LIN {X 0,Y 202.903,Z 833.115,A -85,B 0,C 180,E1 -31559.988,E2 -31559.988} C_VEL
LIN {X 0,Y 208.884,Z 836.315,A -85,B 0,C 180,E1 -31563.074,E2 -31563.074} C_VEL
LIN {X 0,Y 216.378,Z 840.609,A -85,B 0,C 180,E1 -31567.061,E2 -31567.061} C_VEL
LIN {X 0,Y 220.572,Z 843.241,A -85,B 0,C 180,E1 -31569.483,E2 -31569.483} C_VEL
LIN {X 0,Y 224.304,Z 845.645,A -85,B 0,C 180,E1 -31571.741,E2 -31571.741} C_VEL
LIN {X 0,Y 227.405,Z 847.744,A -85,B 0,C 180,E1 -31573.851,E2 -31573.851} C_VEL
LIN {X 0,Y 230.992,Z 850.3,A -85,B 0,C 180,E1 -31576.804,E2 -31576.804} C_VEL
LIN {X 0,Y 235.032,Z 852.777,A -85,B 0,C 180,E1 -31580.667,E2 -31580.667} C_VEL
LIN {X 0,Y 237.24,Z 853.939,A -85,B 0,C 180,E1 -31583.195,E2 -31583.195} C_VEL
LIN {X 0,Y 238.369,Z 854.486,A -85,B 0,C 180,E1 -31584.926,E2 -31584.926} C_VEL
LIN {X 0,Y 239.315,Z 854.891,A -85,B 0,C 180,E1 -31586.829,E2 -31586.829} C_VEL
LIN {X 0,Y 239.828,Z 855.055,A -85,B 0,C 180,E1 -31588.321,E2 -31588.321} C_VEL
LIN {X 0,Y 240.028,Z 855.12,A -85,B 0,C 180,E1 -31590,E2 -31590} C_VEL
LIN {X 0,Y 239.805,Z 855.053,A -85,B 0,C 180,E1 -31591.679,E2 -31591.679} C_VEL
LIN {X 0,Y 239.195,Z 854.848,A -85,B 0,C 180,E1 -31593.369,E2 -31593.369} C_VEL
LIN {X 0,Y 238.362,Z 854.475,A -85,B 0,C 180,E1 -31595.075,E2 -31595.075} C_VEL
LIN {X 0,Y 237.219,Z 853.929,A -85,B 0,C 180,E1 -31596.806,E2 -31596.806} C_VEL
LIN {X 0,Y 235.033,Z 852.788,A -85,B 0,C 180,E1 -31599.335,E2 -31599.335} C_VEL
LIN {X 0,Y 230.986,Z 850.298,A -85,B 0,C 180,E1 -31603.19,E2 -31603.19} C_VEL
LIN {X 0,Y 227.067,Z 847.531,A -85,B 0,C 180,E1 -31606.368,E2 -31606.368} C_VEL
LIN {X 0,Y 223.04,Z 844.829,A -85,B 0,C 180,E1 -31609.041,E2 -31609.041} C_VEL
LIN {X 0,Y 220.517,Z 843.221,A -85,B 0,C 180,E1 -31610.538,E2 -31610.538} C_VEL
LIN {X 0,Y 217.608,Z 841.994,A -85,B 0,C 180,E1 -31611.838,E2 -31611.838} C_VEL
LIN {X 0,Y 213.839,Z 841.077,A -85,B 0,C 180,E1 -31613.032,E2 -31613.032} C_VEL
LIN {X 0,Y 203.07,Z 838.775,A -85,B 0,C 180,E1 -31616.24,E2 -31616.24} C_VEL
LIN {X 0,Y 200.951,Z 837.913,A -85,B 0,C 180,E1 -31617.173,E2 -31617.173} C_VEL
LIN {X 0,Y 194.952,Z 834.972,A -85,B 0,C 180,E1 -31620.31,E2 -31620.31} C_VEL
LIN {X 0,Y 187.377,Z 831.364,A -85,B 0,C 180,E1 -31624.397,E2 -31624.397} C_VEL
LIN {X 0,Y 176.623,Z 826.157,A -85,B 0,C 180,E1 -31630.886,E2 -31630.886} C_VEL
LIN {X 0,Y 162.798,Z 817.399,A -85,B 0,C 180,E1 -31642.817,E2 -31642.817} C_VEL
LIN {X 0,Y 160.588,Z 818.703,A -85,B 0,C 180,E1 -31642.859,E2 -31642.859} C_VEL
LIN {X 0,Y 146.717,Z 829.238,A -85,B 0,C 180,E1 -31640.033,E2 -31640.033} C_VEL
LIN {X 0,Y 134.403,Z 837.203,A -85,B 0,C 180,E1 -31637.058,E2 -31637.058} C_VEL
LIN {X 0,Y 122.45,Z 843.857,A -85,B 0,C 180,E1 -31633.529,E2 -31633.529} C_VEL
LIN {X 0,Y 111.056,Z 849.379,A -85,B 0,C 180,E1 -31629.258,E2 -31629.258} C_VEL
LIN {X 0,Y 100.44,Z 853.782,A -85,B 0,C 180,E1 -31624.039,E2 -31624.039} C_VEL
LIN {X 0,Y 90.867,Z 857.174,A -85,B 0,C 180,E1 -31617.649,E2 -31617.649} C_VEL
LIN {X 0,Y 81.549,Z 859.864,A -85,B 0,C 180,E1 -31608.564,E2 -31608.564} C_VEL
LIN {X 0,Y 76.46,Z 861.04,A -85,B 0,C 180,E1 -31600.593,E2 -31600.593} C_VEL
LIN {X 0,Y 72.976,Z 861.583,A -85,B 0,C 180,E1 -31590,E2 -31590} C_VEL
LIN {X 0,Y 76.461,Z 861.04,A -85,B 0,C 180,E1 -31579.407,E2 -31579.407} C_VEL
LIN {X 0,Y 82.645,Z 859.587,A -85,B 0,C 180,E1 -31570.114,E2 -31570.114} C_VEL
LIN {X 0,Y 90.866,Z 857.173,A -85,B 0,C 180,E1 -31562.351,E2 -31562.351} C_VEL
LIN {X 0,Y 100.444,Z 853.782,A -85,B 0,C 180,E1 -31555.962,E2 -31555.962} C_VEL
LIN {X 0,Y 111.054,Z 849.379,A -85,B 0,C 180,E1 -31550.741,E2 -31550.741} C_VEL
LIN {X 0,Y 122.424,Z 843.858,A -85,B 0,C 180,E1 -31546.459,E2 -31546.459} C_VEL
LIN {X 0,Y 134.403,Z 837.203,A -85,B 0,C 180,E1 -31542.941,E2 -31542.941} C_VEL
LIN {X 0,Y 146.733,Z 829.238,A -85,B 0,C 180,E1 -31539.975,E2 -31539.975} C_VEL
LIN {X 0,Y 160.605,Z 818.703,A -85,B 0,C 180,E1 -31537.149,E2 -31537.149} C_VEL
LIN {X 0,Y 162.798,Z 817.399,A -85,B 0,C 180,E1 -31537.183,E2 -31537.183} C_VEL
LIN {X 0,Y 176.609,Z 826.17,A -85,B 0,C 180,E1 -31549.119,E2 -31549.119} C_VEL
LIN {X 0,Y 187.851,Z 831.576,A -85,B 0,C 180,E1 -31555.863,E2 -31555.863} C_VEL
LIN {X 0,Y 195.144,Z 835.087,A -85,B 0,C 180,E1 -31559.806,E2 -31559.806} C_VEL
LIN {X 0,Y 201.261,Z 838.095,A -85,B 0,C 180,E1 -31563.003,E2 -31563.003} C_VEL
LIN {X 0,Y 209.419,Z 842.368,A -85,B 0,C 180,E1 -31567.349,E2 -31567.349} C_VEL
LIN {X 0,Y 215.586,Z 845.919,A -85,B 0,C 180,E1 -31570.975,E2 -31570.975} C_VEL
LIN {X 0,Y 219.709,Z 848.454,A -85,B 0,C 180,E1 -31573.662,E2 -31573.662} C_VEL
LIN {X 0,Y 224.303,Z 851.529,A -85,B 0,C 180,E1 -31577.331,E2 -31577.331} C_VEL
LIN {X 0,Y 227.865,Z 853.75,A -85,B 0,C 180,E1 -31580.736,E2 -31580.736} C_VEL
LIN {X 0,Y 229.868,Z 854.802,A -85,B 0,C 180,E1 -31582.976,E2 -31582.976} C_VEL
LIN {X 0,Y 231.161,Z 855.444,A -85,B 0,C 180,E1 -31584.767,E2 -31584.767} C_VEL
LIN {X 0,Y 232.263,Z 855.927,A -85,B 0,C 180,E1 -31586.891,E2 -31586.891} C_VEL
LIN {X 0,Y 232.778,Z 856.084,A -85,B 0,C 180,E1 -31588.27,E2 -31588.27} C_VEL
LIN {X 0,Y 233.006,Z 856.158,A -85,B 0,C 180,E1 -31590,E2 -31590} C_VEL
LIN {X 0,Y 232.759,Z 856.085,A -85,B 0,C 180,E1 -31591.73,E2 -31591.73} C_VEL
LIN {X 0,Y 232.081,Z 855.86,A -85,B 0,C 180,E1 -31593.472,E2 -31593.472} C_VEL
LIN {X 0,Y 231.152,Z 855.444,A -85,B 0,C 180,E1 -31595.233,E2 -31595.233} C_VEL
LIN {X 0,Y 229.854,Z 854.809,A -85,B 0,C 180,E1 -31597.025,E2 -31597.025} C_VEL
LIN {X 0,Y 227.867,Z 853.762,A -85,B 0,C 180,E1 -31599.267,E2 -31599.267} C_VEL
LIN {X 0,Y 224.289,Z 851.528,A -85,B 0,C 180,E1 -31602.67,E2 -31602.67} C_VEL
LIN {X 0,Y 219.695,Z 848.469,A -85,B 0,C 180,E1 -31606.326,E2 -31606.326} C_VEL
LIN {X 0,Y 215.549,Z 845.92,A -85,B 0,C 180,E1 -31609.029,E2 -31609.029} C_VEL
LIN {X 0,Y 209.405,Z 842.382,A -85,B 0,C 180,E1 -31612.641,E2 -31612.641} C_VEL
LIN {X 0,Y 200.951,Z 837.913,A -85,B 0,C 180,E1 -31617.173,E2 -31617.173} C_VEL
LIN {X 0,Y 197.626,Z 836.788,A -85,B 0,C 180,E1 -31618.533,E2 -31618.533} C_VEL
LIN {X 0,Y 190.664,Z 835.781,A -85,B 0,C 180,E1 -31620.593,E2 -31620.593} C_VEL
LIN {X 0,Y 184.942,Z 835.104,A -85,B 0,C 180,E1 -31622.296,E2 -31622.296} C_VEL
LIN {X 0,Y 181.269,Z 834.289,A -85,B 0,C 180,E1 -31623.747,E2 -31623.747} C_VEL
LIN {X 0,Y 180.266,Z 833.88,A -85,B 0,C 180,E1 -31624.278,E2 -31624.278} C_VEL
LIN {X 0,Y 172.251,Z 830.257,A -85,B 0,C 180,E1 -31629.177,E2 -31629.177} C_VEL
LIN {X 0,Y 159.808,Z 823.458,A -85,B 0,C 180,E1 -31639.177,E2 -31639.177} C_VEL
LIN {X 0,Y 157.5,Z 824.5,A -85,B 0,C 180,E1 -31639.338,E2 -31639.338} C_VEL
LIN {X 0,Y 145.363,Z 833.226,A -85,B 0,C 180,E1 -31636.486,E2 -31636.486} C_VEL
LIN {X 0,Y 133.54,Z 840.53,A -85,B 0,C 180,E1 -31633.169,E2 -31633.169} C_VEL
LIN {X 0,Y 122.185,Z 846.563,A -85,B 0,C 180,E1 -31629.249,E2 -31629.249} C_VEL
LIN {X 0,Y 109.682,Z 852.261,A -85,B 0,C 180,E1 -31623.595,E2 -31623.595} C_VEL
LIN {X 0,Y 97.33,Z 856.961,A -85,B 0,C 180,E1 -31615.673,E2 -31615.673} C_VEL
LIN {X 0,Y 87.937,Z 859.783,A -85,B 0,C 180,E1 -31606.458,E2 -31606.458} C_VEL
LIN {X 0,Y 83.554,Z 860.825,A -85,B 0,C 180,E1 -31599.684,E2 -31599.684} C_VEL
LIN {X 0,Y 80.137,Z 861.372,A -85,B 0,C 180,E1 -31590,E2 -31590} C_VEL
LIN {X 0,Y 83.555,Z 860.825,A -85,B 0,C 180,E1 -31580.316,E2 -31580.316} C_VEL
LIN {X 0,Y 89.45,Z 859.373,A -85,B 0,C 180,E1 -31571.683,E2 -31571.683} C_VEL
LIN {X 0,Y 97.33,Z 856.961,A -85,B 0,C 180,E1 -31564.327,E2 -31564.327} C_VEL
LIN {X 0,Y 109.68,Z 852.262,A -85,B 0,C 180,E1 -31556.406,E2 -31556.406} C_VEL
LIN {X 0,Y 122.173,Z 846.563,A -85,B 0,C 180,E1 -31550.746,E2 -31550.746} C_VEL
LIN {X 0,Y 136.64,Z 838.692,A -85,B 0,C 180,E1 -31545.901,E2 -31545.901} C_VEL
LIN {X 0,Y 148.422,Z 831.14,A -85,B 0,C 180,E1 -31542.783,E2 -31542.783} C_VEL
LIN {X 0,Y 157.533,Z 824.499,A -85,B 0,C 180,E1 -31540.677,E2 -31540.677} C_VEL
LIN {X 0,Y 159.823,Z 823.457,A -85,B 0,C 180,E1 -31540.829,E2 -31540.829} C_VEL
LIN {X 0,Y 172.239,Z 830.268,A -85,B 0,C 180,E1 -31550.828,E2 -31550.828} C_VEL
LIN {X 0,Y 183.391,Z 835.249,A -85,B 0,C 180,E1 -31557.467,E2 -31557.467} C_VEL
LIN {X 0,Y 191.402,Z 838.842,A -85,B 0,C 180,E1 -31561.791,E2 -31561.791} C_VEL
LIN {X 0,Y 196.719,Z 841.243,A -85,B 0,C 180,E1 -31564.615,E2 -31564.615} C_VEL
LIN {X 0,Y 203.902,Z 844.75,A -85,B 0,C 180,E1 -31568.53,E2 -31568.53} C_VEL
LIN {X 0,Y 208.106,Z 846.961,A -85,B 0,C 180,E1 -31571.011,E2 -31571.011} C_VEL
LIN {X 0,Y 212.316,Z 849.306,A -85,B 0,C 180,E1 -31573.726,E2 -31573.726} C_VEL
LIN {X 0,Y 216.441,Z 851.835,A -85,B 0,C 180,E1 -31576.934,E2 -31576.934} C_VEL
LIN {X 0,Y 218.611,Z 853.231,A -85,B 0,C 180,E1 -31578.879,E2 -31578.879} C_VEL
LIN {X 0,Y 220.68,Z 854.365,A -85,B 0,C 180,E1 -31580.838,E2 -31580.838} C_VEL
LIN {X 0,Y 222.416,Z 855.312,A -85,B 0,C 180,E1 -31582.739,E2 -31582.739} C_VEL
LIN {X 0,Y 223.851,Z 856.031,A -85,B 0,C 180,E1 -31584.596,E2 -31584.596} C_VEL
LIN {X 0,Y 225.207,Z 856.635,A -85,B 0,C 180,E1 -31586.975,E2 -31586.975} C_VEL
LIN {X 0,Y 225.66,Z 856.792,A -85,B 0,C 180,E1 -31588.215,E2 -31588.215} C_VEL
LIN {X 0,Y 225.935,Z 856.875,A -85,B 0,C 180,E1 -31590,E2 -31590} C_VEL
LIN {X 0,Y 225.644,Z 856.796,A -85,B 0,C 180,E1 -31591.785,E2 -31591.785} C_VEL
LIN {X 0,Y 224.902,Z 856.532,A -85,B 0,C 180,E1 -31593.583,E2 -31593.583} C_VEL
LIN {X 0,Y 223.842,Z 856.039,A -85,B 0,C 180,E1 -31595.405,E2 -31595.405} C_VEL
LIN {X 0,Y 222.405,Z 855.308,A -85,B 0,C 180,E1 -31597.261,E2 -31597.261} C_VEL
LIN {X 0,Y 220.68,Z 854.366,A -85,B 0,C 180,E1 -31599.162,E2 -31599.162} C_VEL
LIN {X 0,Y 218.613,Z 853.231,A -85,B 0,C 180,E1 -31601.121,E2 -31601.121} C_VEL
LIN {X 0,Y 216.341,Z 851.781,A -85,B 0,C 180,E1 -31603.144,E2 -31603.144} C_VEL
LIN {X 0,Y 212.307,Z 849.314,A -85,B 0,C 180,E1 -31606.266,E2 -31606.266} C_VEL
LIN {X 0,Y 208.098,Z 846.969,A -85,B 0,C 180,E1 -31608.983,E2 -31608.983} C_VEL
LIN {X 0,Y 202.014,Z 843.832,A -85,B 0,C 180,E1 -31612.5,E2 -31612.5} C_VEL
LIN {X 0,Y 194.896,Z 840.388,A -85,B 0,C 180,E1 -31616.354,E2 -31616.354} C_VEL
LIN {X 0,Y 187.335,Z 836.998,A -85,B 0,C 180,E1 -31620.362,E2 -31620.362} C_VEL
LIN {X 0,Y 180.266,Z 833.88,A -85,B 0,C 180,E1 -31624.278,E2 -31624.278} C_VEL
LIN {X 0,Y 176.99,Z 832.953,A -85,B 0,C 180,E1 -31625.821,E2 -31625.821} C_VEL
LIN {X 0,Y 170.275,Z 832.301,A -85,B 0,C 180,E1 -31628.215,E2 -31628.215} C_VEL
LIN {X 0,Y 164.882,Z 831.868,A -85,B 0,C 180,E1 -31630.224,E2 -31630.224} C_VEL
LIN {X 0,Y 161.52,Z 831.172,A -85,B 0,C 180,E1 -31631.928,E2 -31631.928} C_VEL
LIN {X 0,Y 160.634,Z 830.815,A -85,B 0,C 180,E1 -31632.546,E2 -31632.546} C_VEL
LIN {X 0,Y 156.751,Z 828.796,A -85,B 0,C 180,E1 -31635.836,E2 -31635.836} C_VEL
LIN {X 0,Y 156.312,Z 828.815,A -85,B 0,C 180,E1 -31636.002,E2 -31636.002} C_VEL
LIN {X 0,Y 144.598,Z 836.785,A -85,B 0,C 180,E1 -31632.878,E2 -31632.878} C_VEL
LIN {X 0,Y 133.295,Z 843.432,A -85,B 0,C 180,E1 -31629.249,E2 -31629.249} C_VEL
LIN {X 0,Y 122.573,Z 848.958,A -85,B 0,C 180,E1 -31624.985,E2 -31624.985} C_VEL
LIN {X 0,Y 112.704,Z 853.353,A -85,B 0,C 180,E1 -31619.924,E2 -31619.924} C_VEL
LIN {X 0,Y 103.892,Z 856.748,A -85,B 0,C 180,E1 -31613.946,E2 -31613.946} C_VEL
LIN {X 0,Y 94.435,Z 859.688,A -85,B 0,C 180,E1 -31604.657,E2 -31604.657} C_VEL
LIN {X 0,Y 88.689,Z 860.946,A -85,B 0,C 180,E1 -31594.545,E2 -31594.545} C_VEL
LIN {X 0,Y 87.31,Z 861.16,A -85,B 0,C 180,E1 -31590,E2 -31590} C_VEL
LIN {X 0,Y 90.667,Z 860.611,A -85,B 0,C 180,E1 -31581.082,E2 -31581.082} C_VEL
LIN {X 0,Y 96.321,Z 859.158,A -85,B 0,C 180,E1 -31573.031,E2 -31573.031} C_VEL
LIN {X 0,Y 103.893,Z 856.748,A -85,B 0,C 180,E1 -31566.054,E2 -31566.054} C_VEL
LIN {X 0,Y 115.065,Z 852.356,A -85,B 0,C 180,E1 -31558.768,E2 -31558.768} C_VEL
LIN {X 0,Y 125.186,Z 847.669,A -85,B 0,C 180,E1 -31553.881,E2 -31553.881} C_VEL
LIN {X 0,Y 136.047,Z 841.889,A -85,B 0,C 180,E1 -31549.781,E2 -31549.781} C_VEL
LIN {X 0,Y 147.492,Z 834.947,A -85,B 0,C 180,E1 -31546.298,E2 -31546.298} C_VEL
LIN {X 0,Y 156.329,Z 828.814,A -85,B 0,C 180,E1 -31544.004,E2 -31544.004} C_VEL
LIN {X 0,Y 156.733,Z 828.797,A -85,B 0,C 180,E1 -31544.157,E2 -31544.157} C_VEL
LIN {X 0,Y 167.935,Z 834.178,A -85,B 0,C 180,E1 -31552.667,E2 -31552.667} C_VEL
LIN {X 0,Y 175.515,Z 837.267,A -85,B 0,C 180,E1 -31557.232,E2 -31557.232} C_VEL
LIN {X 0,Y 183.577,Z 840.555,A -85,B 0,C 180,E1 -31561.704,E2 -31561.704} C_VEL
LIN {X 0,Y 187.76,Z 842.305,A -85,B 0,C 180,E1 -31563.938,E2 -31563.938} C_VEL
LIN {X 0,Y 192.07,Z 844.153,A -85,B 0,C 180,E1 -31566.266,E2 -31566.266} C_VEL
LIN {X 0,Y 197.335,Z 846.497,A -85,B 0,C 180,E1 -31569.137,E2 -31569.137} C_VEL
LIN {X 0,Y 201.689,Z 848.569,A -85,B 0,C 180,E1 -31571.723,E2 -31571.723} C_VEL
LIN {X 0,Y 205.35,Z 850.388,A -85,B 0,C 180,E1 -31574.11,E2 -31574.11} C_VEL
LIN {X 0,Y 209.141,Z 852.488,A -85,B 0,C 180,E1 -31577.034,E2 -31577.034} C_VEL
LIN {X 0,Y 210.783,Z 853.466,A -85,B 0,C 180,E1 -31578.46,E2 -31578.46} C_VEL
LIN {X 0,Y 213.479,Z 854.859,A -85,B 0,C 180,E1 -31580.976,E2 -31580.976} C_VEL
LIN {X 0,Y 214.893,Z 855.555,A -85,B 0,C 180,E1 -31582.483,E2 -31582.483} C_VEL
LIN {X 0,Y 216.462,Z 856.339,A -85,B 0,C 180,E1 -31584.411,E2 -31584.411} C_VEL
LIN {X 0,Y 218.14,Z 857.02,A -85,B 0,C 180,E1 -31587.121,E2 -31587.121} C_VEL
LIN {X 0,Y 218.854,Z 857.272,A -85,B 0,C 180,E1 -31590,E2 -31590} C_VEL
LIN {X 0,Y 218.136,Z 857.025,A -85,B 0,C 180,E1 -31592.858,E2 -31592.858} C_VEL
LIN {X 0,Y 216.453,Z 856.339,A -85,B 0,C 180,E1 -31595.59,E2 -31595.59} C_VEL
LIN {X 0,Y 214.887,Z 855.556,A -85,B 0,C 180,E1 -31597.517,E2 -31597.517} C_VEL
LIN {X 0,Y 212.969,Z 854.598,A -85,B 0,C 180,E1 -31599.497,E2 -31599.497} C_VEL
LIN {X 0,Y 210.783,Z 853.466,A -85,B 0,C 180,E1 -31601.54,E2 -31601.54} C_VEL
LIN {X 0,Y 208.237,Z 852.026,A -85,B 0,C 180,E1 -31603.665,E2 -31603.665} C_VEL
LIN {X 0,Y 204.905,Z 850.162,A -85,B 0,C 180,E1 -31606.188,E2 -31606.188} C_VEL
LIN {X 0,Y 200.599,Z 848.03,A -85,B 0,C 180,E1 -31608.927,E2 -31608.927} C_VEL
LIN {X 0,Y 196.286,Z 846.05,A -85,B 0,C 180,E1 -31611.422,E2 -31611.422} C_VEL
LIN {X 0,Y 191.988,Z 844.124,A -85,B 0,C 180,E1 -31613.774,E2 -31613.774} C_VEL
LIN {X 0,Y 186.112,Z 841.59,A -85,B 0,C 180,E1 -31616.945,E2 -31616.945} C_VEL
LIN {X 0,Y 179.298,Z 838.839,A -85,B 0,C 180,E1 -31620.634,E2 -31620.634} C_VEL
LIN {X 0,Y 171.662,Z 835.698,A -85,B 0,C 180,E1 -31625.035,E2 -31625.035} C_VEL
LIN {X 0,Y 160.634,Z 830.815,A -85,B 0,C 180,E1 -31632.546,E2 -31632.546} C_VEL
LIN {X 0,Y 159.568,Z 830.875,A -85,B 0,C 180,E1 -31632.887,E2 -31632.887} C_VEL
LIN {X 0,Y 157.126,Z 831.782,A -85,B 0,C 180,E1 -31632.998,E2 -31632.998} C_VEL
LIN {X 0,Y 153.935,Z 833.506,A -85,B 0,C 180,E1 -31632.595,E2 -31632.595} C_VEL
LIN {X 0,Y 148.459,Z 837.36,A -85,B 0,C 180,E1 -31630.799,E2 -31630.799} C_VEL
LIN {X 0,Y 143.925,Z 840.362,A -85,B 0,C 180,E1 -31629.105,E2 -31629.105} C_VEL
LIN {X 0,Y 133.687,Z 846.134,A -85,B 0,C 180,E1 -31625.328,E2 -31625.328} C_VEL
LIN {X 0,Y 123.661,Z 851.081,A -85,B 0,C 180,E1 -31620.763,E2 -31620.763} C_VEL
LIN {X 0,Y 114.61,Z 854.929,A -85,B 0,C 180,E1 -31615.419,E2 -31615.419} C_VEL
LIN {X 0,Y 106.713,Z 857.827,A -85,B 0,C 180,E1 -31609.225,E2 -31609.225} C_VEL
LIN {X 0,Y 100.286,Z 859.76,A -85,B 0,C 180,E1 -31602.136,E2 -31602.136} C_VEL
LIN {X 0,Y 95.842,Z 860.737,A -85,B 0,C 180,E1 -31594.205,E2 -31594.205} C_VEL
LIN {X 0,Y 94.494,Z 860.947,A -85,B 0,C 180,E1 -31590,E2 -31590} C_VEL
LIN {X 0,Y 97.796,Z 860.396,A -85,B 0,C 180,E1 -31581.737,E2 -31581.737} C_VEL
LIN {X 0,Y 103.268,Z 858.942,A -85,B 0,C 180,E1 -31574.204,E2 -31574.204} C_VEL
LIN {X 0,Y 110.534,Z 856.536,A -85,B 0,C 180,E1 -31567.574,E2 -31567.574} C_VEL
LIN {X 0,Y 120.694,Z 852.41,A -85,B 0,C 180,E1 -31560.86,E2 -31560.86} C_VEL
LIN {X 0,Y 131.092,Z 847.459,A -85,B 0,C 180,E1 -31555.743,E2 -31555.743} C_VEL
LIN {X 0,Y 141.642,Z 841.678,A -85,B 0,C 180,E1 -31551.669,E2 -31551.669} C_VEL
LIN {X 0,Y 152.464,Z 834.953,A -85,B 0,C 180,E1 -31548.26,E2 -31548.26} C_VEL
LIN {X 0,Y 154.544,Z 833.994,A -85,B 0,C 180,E1 -31548.109,E2 -31548.109} C_VEL
LIN {X 0,Y 167.591,Z 839.291,A -85,B 0,C 180,E1 -31557.002,E2 -31557.002} C_VEL
LIN {X 0,Y 175.719,Z 842.283,A -85,B 0,C 180,E1 -31561.629,E2 -31561.629} C_VEL
LIN {X 0,Y 181.627,Z 844.494,A -85,B 0,C 180,E1 -31564.809,E2 -31564.809} C_VEL
LIN {X 0,Y 188.623,Z 847.294,A -85,B 0,C 180,E1 -31568.665,E2 -31568.665} C_VEL
LIN {X 0,Y 193.066,Z 849.118,A -85,B 0,C 180,E1 -31571.162,E2 -31571.162} C_VEL
LIN {X 0,Y 197.474,Z 851.04,A -85,B 0,C 180,E1 -31573.925,E2 -31573.925} C_VEL
LIN {X 0,Y 201.831,Z 853.152,A -85,B 0,C 180,E1 -31577.156,E2 -31577.156} C_VEL
LIN {X 0,Y 206.282,Z 855.342,A -85,B 0,C 180,E1 -31581.119,E2 -31581.119} C_VEL
LIN {X 0,Y 209.018,Z 856.557,A -85,B 0,C 180,E1 -31584.211,E2 -31584.211} C_VEL
LIN {X 0,Y 211.075,Z 857.269,A -85,B 0,C 180,E1 -31587.276,E2 -31587.276} C_VEL
LIN {X 0,Y 211.75,Z 857.482,A -85,B 0,C 180,E1 -31590,E2 -31590} C_VEL
LIN {X 0,Y 211.072,Z 857.271,A -85,B 0,C 180,E1 -31592.706,E2 -31592.706} C_VEL
LIN {X 0,Y 209.011,Z 856.557,A -85,B 0,C 180,E1 -31595.789,E2 -31595.789} C_VEL
LIN {X 0,Y 206.282,Z 855.343,A -85,B 0,C 180,E1 -31598.881,E2 -31598.881} C_VEL
LIN {X 0,Y 201.828,Z 853.156,A -85,B 0,C 180,E1 -31602.84,E2 -31602.84} C_VEL
LIN {X 0,Y 197.467,Z 851.047,A -85,B 0,C 180,E1 -31606.068,E2 -31606.068} C_VEL
LIN {X 0,Y 192.398,Z 848.861,A -85,B 0,C 180,E1 -31609.193,E2 -31609.193} C_VEL
LIN {X 0,Y 187.349,Z 846.817,A -85,B 0,C 180,E1 -31612.032,E2 -31612.032} C_VEL
LIN {X 0,Y 179.979,Z 843.878,A -85,B 0,C 180,E1 -31616.089,E2 -31616.089} C_VEL
LIN {X 0,Y 171.585,Z 840.751,A -85,B 0,C 180,E1 -31620.669,E2 -31620.669} C_VEL
LIN {X 0,Y 163.737,Z 837.799,A -85,B 0,C 180,E1 -31625.362,E2 -31625.362} C_VEL
LIN {X 0,Y 154.544,Z 833.987,A -85,B 0,C 180,E1 -31631.897,E2 -31631.897} C_VEL
LIN {X 0,Y 152.464,Z 834.942,A -85,B 0,C 180,E1 -31631.75,E2 -31631.75} C_VEL
LIN {X 0,Y 143.925,Z 840.362,A -85,B 0,C 180,E1 -31629.105,E2 -31629.105} C_VEL
LIN {X 0,Y 140.3,Z 842.755,A -85,B 0,C 180,E1 -31627.479,E2 -31627.479} C_VEL
LIN {X 0,Y 132.687,Z 849.09,A -85,B 0,C 180,E1 -31621.236,E2 -31621.236} C_VEL
LIN {X 0,Y 129.812,Z 850.892,A -85,B 0,C 180,E1 -31619.127,E2 -31619.127} C_VEL
LIN {X 0,Y 128.668,Z 851.442,A -85,B 0,C 180,E1 -31618.463,E2 -31618.463} C_VEL
LIN {X 0,Y 117.24,Z 856.323,A -85,B 0,C 180,E1 -31611.08,E2 -31611.08} C_VEL
LIN {X 0,Y 110.272,Z 858.726,A -85,B 0,C 180,E1 -31604.769,E2 -31604.769} C_VEL
LIN {X 0,Y 104.932,Z 860.182,A -85,B 0,C 180,E1 -31597.698,E2 -31597.698} C_VEL
LIN {X 0,Y 101.676,Z 860.735,A -85,B 0,C 180,E1 -31590,E2 -31590} C_VEL
LIN {X 0,Y 104.932,Z 860.182,A -85,B 0,C 180,E1 -31582.302,E2 -31582.302} C_VEL
LIN {X 0,Y 110.223,Z 858.727,A -85,B 0,C 180,E1 -31575.224,E2 -31575.224} C_VEL
LIN {X 0,Y 117.242,Z 856.323,A -85,B 0,C 180,E1 -31568.921,E2 -31568.921} C_VEL
LIN {X 0,Y 126.463,Z 852.464,A -85,B 0,C 180,E1 -31562.768,E2 -31562.768} C_VEL
LIN {X 0,Y 137.111,Z 847.249,A -85,B 0,C 180,E1 -31557.439,E2 -31557.439} C_VEL
LIN {X 0,Y 147.367,Z 841.466,A -85,B 0,C 180,E1 -31553.408,E2 -31553.408} C_VEL
LIN {X 0,Y 151.841,Z 838.728,A -85,B 0,C 180,E1 -31551.89,E2 -31551.89} C_VEL
LIN {X 0,Y 155.78,Z 839.883,A -85,B 0,C 180,E1 -31554.297,E2 -31554.297} C_VEL
LIN {X 0,Y 163.634,Z 842.573,A -85,B 0,C 180,E1 -31559.202,E2 -31559.202} C_VEL
LIN {X 0,Y 172.116,Z 845.419,A -85,B 0,C 180,E1 -31563.937,E2 -31563.937} C_VEL
LIN {X 0,Y 177.015,Z 847.147,A -85,B 0,C 180,E1 -31566.608,E2 -31566.608} C_VEL
LIN {X 0,Y 182.696,Z 849.168,A -85,B 0,C 180,E1 -31569.745,E2 -31569.745} C_VEL
LIN {X 0,Y 187.573,Z 850.939,A -85,B 0,C 180,E1 -31572.558,E2 -31572.558} C_VEL
LIN {X 0,Y 191.545,Z 852.533,A -85,B 0,C 180,E1 -31575.118,E2 -31575.118} C_VEL
LIN {X 0,Y 194.781,Z 853.947,A -85,B 0,C 180,E1 -31577.497,E2 -31577.497} C_VEL
LIN {X 0,Y 199.077,Z 855.79,A -85,B 0,C 180,E1 -31581.29,E2 -31581.29} C_VEL
LIN {X 0,Y 201.541,Z 856.776,A -85,B 0,C 180,E1 -31583.995,E2 -31583.995} C_VEL
LIN {X 0,Y 204.005,Z 857.506,A -85,B 0,C 180,E1 -31587.489,E2 -31587.489} C_VEL
LIN {X 0,Y 204.644,Z 857.692,A -85,B 0,C 180,E1 -31590,E2 -31590} C_VEL
LIN {X 0,Y 204.002,Z 857.507,A -85,B 0,C 180,E1 -31592.494,E2 -31592.494} C_VEL
LIN {X 0,Y 201.536,Z 856.776,A -85,B 0,C 180,E1 -31596.005,E2 -31596.005} C_VEL
LIN {X 0,Y 199.077,Z 855.79,A -85,B 0,C 180,E1 -31598.71,E2 -31598.71} C_VEL
LIN {X 0,Y 194.507,Z 853.832,A -85,B 0,C 180,E1 -31602.693,E2 -31602.693} C_VEL
LIN {X 0,Y 190.02,Z 851.935,A -85,B 0,C 180,E1 -31605.927,E2 -31605.927} C_VEL
LIN {X 0,Y 185.459,Z 850.174,A -85,B 0,C 180,E1 -31608.672,E2 -31608.672} C_VEL
LIN {X 0,Y 180.937,Z 848.522,A -85,B 0,C 180,E1 -31611.22,E2 -31611.22} C_VEL
LIN {X 0,Y 176.511,Z 846.946,A -85,B 0,C 180,E1 -31613.686,E2 -31613.686} C_VEL
LIN {X 0,Y 167.825,Z 844.012,A -85,B 0,C 180,E1 -31618.43,E2 -31618.43} C_VEL
LIN {X 0,Y 159.624,Z 841.188,A -85,B 0,C 180,E1 -31623.225,E2 -31623.225} C_VEL
LIN {X 0,Y 155.311,Z 839.692,A -85,B 0,C 180,E1 -31626.033,E2 -31626.033} C_VEL
LIN {X 0,Y 151.845,Z 838.726,A -85,B 0,C 180,E1 -31628.111,E2 -31628.111} C_VEL
LIN {X 0,Y 139.643,Z 845.92,A -85,B 0,C 180,E1 -31623.614,E2 -31623.614} C_VEL
LIN {X 0,Y 128.668,Z 851.442,A -85,B 0,C 180,E1 -31618.463,E2 -31618.463} C_VEL
LIN {X 0,Y 125.679,Z 853.079,A -85,B 0,C 180,E1 -31616.28,E2 -31616.28} C_VEL
LIN {X 0,Y 122.718,Z 855.332,A -85,B 0,C 180,E1 -31612.04,E2 -31612.04} C_VEL
LIN {X 0,Y 120.934,Z 856.879,A -85,B 0,C 180,E1 -31608.47,E2 -31608.47} C_VEL
LIN {X 0,Y 119.134,Z 857.844,A -85,B 0,C 180,E1 -31605.825,E2 -31605.825} C_VEL
LIN {X 0,Y 118.339,Z 858.125,A -85,B 0,C 180,E1 -31604.968,E2 -31604.968} C_VEL
LIN {X 0,Y 112.067,Z 859.968,A -85,B 0,C 180,E1 -31597.205,E2 -31597.205} C_VEL
LIN {X 0,Y 108.856,Z 860.523,A -85,B 0,C 180,E1 -31590,E2 -31590} C_VEL
LIN {X 0,Y 112.068,Z 859.968,A -85,B 0,C 180,E1 -31582.795,E2 -31582.795} C_VEL
LIN {X 0,Y 117.226,Z 858.512,A -85,B 0,C 180,E1 -31576.125,E2 -31576.125} C_VEL
LIN {X 0,Y 124,Z 856.111,A -85,B 0,C 180,E1 -31570.12,E2 -31570.12} C_VEL
LIN {X 0,Y 132.346,Z 852.511,A -85,B 0,C 180,E1 -31564.521,E2 -31564.521} C_VEL
LIN {X 0,Y 143.255,Z 847.038,A -85,B 0,C 180,E1 -31558.995,E2 -31558.995} C_VEL
LIN {X 0,Y 150.76,Z 842.793,A -85,B 0,C 180,E1 -31555.986,E2 -31555.986} C_VEL
LIN {X 0,Y 159.858,Z 845.637,A -85,B 0,C 180,E1 -31561.553,E2 -31561.553} C_VEL
LIN {X 0,Y 166.026,Z 847.501,A -85,B 0,C 180,E1 -31564.957,E2 -31564.957} C_VEL
LIN {X 0,Y 173.229,Z 849.746,A -85,B 0,C 180,E1 -31568.924,E2 -31568.924} C_VEL
LIN {X 0,Y 177.995,Z 851.238,A -85,B 0,C 180,E1 -31571.587,E2 -31571.587} C_VEL
LIN {X 0,Y 182.702,Z 852.803,A -85,B 0,C 180,E1 -31574.38,E2 -31574.38} C_VEL
LIN {X 0,Y 187.166,Z 854.48,A -85,B 0,C 180,E1 -31577.494,E2 -31577.494} C_VEL
LIN {X 0,Y 189.356,Z 855.309,A -85,B 0,C 180,E1 -31579.306,E2 -31579.306} C_VEL
LIN {X 0,Y 191.951,Z 856.245,A -85,B 0,C 180,E1 -31581.579,E2 -31581.579} C_VEL
LIN {X 0,Y 193.989,Z 856.997,A -85,B 0,C 180,E1 -31583.761,E2 -31583.761} C_VEL
LIN {X 0,Y 195.682,Z 857.468,A -85,B 0,C 180,E1 -31585.881,E2 -31585.881} C_VEL
LIN {X 0,Y 197.064,Z 857.756,A -85,B 0,C 180,E1 -31587.956,E2 -31587.956} C_VEL
LIN {X 0,Y 197.538,Z 857.902,A -85,B 0,C 180,E1 -31590,E2 -31590} C_VEL
LIN {X 0,Y 196.934,Z 857.742,A -85,B 0,C 180,E1 -31592.26,E2 -31592.26} C_VEL
LIN {X 0,Y 195.679,Z 857.468,A -85,B 0,C 180,E1 -31594.119,E2 -31594.119} C_VEL
LIN {X 0,Y 193.985,Z 856.997,A -85,B 0,C 180,E1 -31596.24,E2 -31596.24} C_VEL
LIN {X 0,Y 191.862,Z 856.218,A -85,B 0,C 180,E1 -31598.503,E2 -31598.503} C_VEL
LIN {X 0,Y 187.162,Z 854.483,A -85,B 0,C 180,E1 -31602.501,E2 -31602.501} C_VEL
LIN {X 0,Y 182.524,Z 852.753,A -85,B 0,C 180,E1 -31605.72,E2 -31605.72} C_VEL
LIN {X 0,Y 177.849,Z 851.196,A -85,B 0,C 180,E1 -31608.489,E2 -31608.489} C_VEL
LIN {X 0,Y 172.386,Z 849.496,A -85,B 0,C 180,E1 -31611.525,E2 -31611.525} C_VEL
LIN {X 0,Y 164.237,Z 846.942,A -85,B 0,C 180,E1 -31616.023,E2 -31616.023} C_VEL
LIN {X 0,Y 155.677,Z 844.378,A -85,B 0,C 180,E1 -31620.937,E2 -31620.937} C_VEL
LIN {X 0,Y 150.689,Z 842.796,A -85,B 0,C 180,E1 -31624.032,E2 -31624.032} C_VEL
LIN {X 0,Y 140.886,Z 848.326,A -85,B 0,C 180,E1 -31619.923,E2 -31619.923} C_VEL
LIN {X 0,Y 131.925,Z 852.709,A -85,B 0,C 180,E1 -31615.225,E2 -31615.225} C_VEL
LIN {X 0,Y 123.998,Z 856.111,A -85,B 0,C 180,E1 -31609.881,E2 -31609.881} C_VEL
LIN {X 0,Y 118.339,Z 858.125,A -85,B 0,C 180,E1 -31604.968,E2 -31604.968} C_VEL
LIN {X 0,Y 115.803,Z 859.184,A -85,B 0,C 180,E1 -31601.348,E2 -31601.348} C_VEL
LIN {X 0,Y 114.857,Z 859.921,A -85,B 0,C 180,E1 -31597.462,E2 -31597.462} C_VEL
LIN {X 0,Y 115.582,Z 860.346,A -85,B 0,C 180,E1 -31591.522,E2 -31591.522} C_VEL
LIN {X 0,Y 116.18,Z 860.285,A -85,B 0,C 180,E1 -31589.57,E2 -31589.57} C_VEL
LIN {X 0,Y 119.211,Z 859.754,A -85,B 0,C 180,E1 -31583.229,E2 -31583.229} C_VEL
LIN {X 0,Y 124.252,Z 858.297,A -85,B 0,C 180,E1 -31576.924,E2 -31576.924} C_VEL
LIN {X 0,Y 130.8,Z 855.899,A -85,B 0,C 180,E1 -31571.193,E2 -31571.193} C_VEL
LIN {X 0,Y 140.564,Z 851.493,A -85,B 0,C 180,E1 -31564.851,E2 -31564.851} C_VEL
LIN {X 0,Y 147.176,Z 848.116,A -85,B 0,C 180,E1 -31561.477,E2 -31561.477} C_VEL
LIN {X 0,Y 150.584,Z 846.888,A -85,B 0,C 180,E1 -31560.779,E2 -31560.779} C_VEL
LIN {X 0,Y 160.853,Z 849.644,A -85,B 0,C 180,E1 -31566.566,E2 -31566.566} C_VEL
LIN {X 0,Y 167.854,Z 851.556,A -85,B 0,C 180,E1 -31570.43,E2 -31570.43} C_VEL
LIN {X 0,Y 174.999,Z 853.585,A -85,B 0,C 180,E1 -31574.543,E2 -31574.543} C_VEL
LIN {X 0,Y 179.812,Z 855.081,A -85,B 0,C 180,E1 -31577.719,E2 -31577.719} C_VEL
LIN {X 0,Y 184.636,Z 856.657,A -85,B 0,C 180,E1 -31581.75,E2 -31581.75} C_VEL
LIN {X 0,Y 186.361,Z 857.221,A -85,B 0,C 180,E1 -31583.504,E2 -31583.504} C_VEL
LIN {X 0,Y 188.233,Z 857.691,A -85,B 0,C 180,E1 -31585.718,E2 -31585.718} C_VEL
LIN {X 0,Y 189.871,Z 857.976,A -85,B 0,C 180,E1 -31587.981,E2 -31587.981} C_VEL
LIN {X 0,Y 190.43,Z 858.112,A -85,B 0,C 180,E1 -31590,E2 -31590} C_VEL
LIN {X 0,Y 189.797,Z 857.97,A -85,B 0,C 180,E1 -31592.122,E2 -31592.122} C_VEL
LIN {X 0,Y 188.23,Z 857.691,A -85,B 0,C 180,E1 -31594.282,E2 -31594.282} C_VEL
LIN {X 0,Y 186.359,Z 857.221,A -85,B 0,C 180,E1 -31596.496,E2 -31596.496} C_VEL
LIN {X 0,Y 184.003,Z 856.485,A -85,B 0,C 180,E1 -31598.788,E2 -31598.788} C_VEL
LIN {X 0,Y 179.809,Z 855.083,A -85,B 0,C 180,E1 -31602.277,E2 -31602.277} C_VEL
LIN {X 0,Y 174.989,Z 853.594,A -85,B 0,C 180,E1 -31605.445,E2 -31605.445} C_VEL
LIN {X 0,Y 167.818,Z 851.557,A -85,B 0,C 180,E1 -31609.574,E2 -31609.574} C_VEL
LIN {X 0,Y 160.855,Z 849.642,A -85,B 0,C 180,E1 -31613.436,E2 -31613.436} C_VEL
LIN {X 0,Y 150.594,Z 846.884,A -85,B 0,C 180,E1 -31619.223,E2 -31619.223} C_VEL
LIN {X 0,Y 147.188,Z 848.116,A -85,B 0,C 180,E1 -31618.521,E2 -31618.521} C_VEL
LIN {X 0,Y 138.354,Z 852.55,A -85,B 0,C 180,E1 -31613.889,E2 -31613.889} C_VEL
LIN {X 0,Y 130.798,Z 855.899,A -85,B 0,C 180,E1 -31608.807,E2 -31608.807} C_VEL
LIN {X 0,Y 124.275,Z 858.296,A -85,B 0,C 180,E1 -31603.074,E2 -31603.074} C_VEL
LIN {X 0,Y 119.211,Z 859.754,A -85,B 0,C 180,E1 -31596.771,E2 -31596.771} C_VEL
LIN {X 0,Y 116.039,Z 860.311,A -85,B 0,C 180,E1 -31590,E2 -31590} C_VEL
LIN {X 0,Y 116.18,Z 860.285,A -85,B 0,C 180,E1 -31589.57,E2 -31589.57} C_VEL
LIN {X 0,Y 117.953,Z 860.104,A -85,B 0,C 180,E1 -31586.813,E2 -31586.813} C_VEL
LIN {X 0,Y 123.19,Z 859.54,A -85,B 0,C 180,E1 -31582.816,E2 -31582.816} C_VEL
LIN {X 0,Y 127.969,Z 858.84,A -85,B 0,C 180,E1 -31579.919,E2 -31579.919} C_VEL
LIN {X 0,Y 131.128,Z 858.112,A -85,B 0,C 180,E1 -31577.719,E2 -31577.719} C_VEL
LIN {X 0,Y 132.001,Z 857.818,A -85,B 0,C 180,E1 -31576.956,E2 -31576.956} C_VEL
LIN {X 0,Y 137.663,Z 855.686,A -85,B 0,C 180,E1 -31572.163,E2 -31572.163} C_VEL
LIN {X 0,Y 147.104,Z 851.292,A -85,B 0,C 180,E1 -31566.054,E2 -31566.054} C_VEL
LIN {X 0,Y 149.201,Z 850.24,A -85,B 0,C 180,E1 -31564.917,E2 -31564.917} C_VEL
LIN {X 0,Y 149.77,Z 850.221,A -85,B 0,C 180,E1 -31565.019,E2 -31565.019} C_VEL
LIN {X 0,Y 157.688,Z 852.058,A -85,B 0,C 180,E1 -31569.379,E2 -31569.379} C_VEL
LIN {X 0,Y 163.298,Z 853.397,A -85,B 0,C 180,E1 -31572.467,E2 -31572.467} C_VEL
LIN {X 0,Y 168.611,Z 854.739,A -85,B 0,C 180,E1 -31575.518,E2 -31575.518} C_VEL
LIN {X 0,Y 172.814,Z 855.809,A -85,B 0,C 180,E1 -31578.268,E2 -31578.268} C_VEL
LIN {X 0,Y 177.419,Z 857.092,A -85,B 0,C 180,E1 -31582.01,E2 -31582.01} C_VEL
LIN {X 0,Y 180.736,Z 857.914,A -85,B 0,C 180,E1 -31585.54,E2 -31585.54} C_VEL
LIN {X 0,Y 182.811,Z 858.21,A -85,B 0,C 180,E1 -31588.24,E2 -31588.24} C_VEL
LIN {X 0,Y 183.296,Z 858.323,A -85,B 0,C 180,E1 -31590,E2 -31590} C_VEL
LIN {X 0,Y 182.811,Z 858.21,A -85,B 0,C 180,E1 -31591.757,E2 -31591.757} C_VEL
LIN {X 0,Y 180.734,Z 857.914,A -85,B 0,C 180,E1 -31594.46,E2 -31594.46} C_VEL
LIN {X 0,Y 178.655,Z 857.447,A -85,B 0,C 180,E1 -31596.777,E2 -31596.777} C_VEL
LIN {X 0,Y 175.951,Z 856.728,A -85,B 0,C 180,E1 -31599.193,E2 -31599.193} C_VEL
LIN {X 0,Y 172.422,Z 855.715,A -85,B 0,C 180,E1 -31601.976,E2 -31601.976} C_VEL
LIN {X 0,Y 167.453,Z 854.438,A -85,B 0,C 180,E1 -31605.139,E2 -31605.139} C_VEL
LIN {X 0,Y 162.526,Z 853.228,A -85,B 0,C 180,E1 -31607.952,E2 -31607.952} C_VEL
LIN {X 0,Y 157.036,Z 851.899,A -85,B 0,C 180,E1 -31610.979,E2 -31610.979} C_VEL
LIN {X 0,Y 149.776,Z 850.221,A -85,B 0,C 180,E1 -31614.98,E2 -31614.98} C_VEL
LIN {X 0,Y 149.206,Z 850.24,A -85,B 0,C 180,E1 -31615.082,E2 -31615.082} C_VEL
LIN {X 0,Y 141.253,Z 854.081,A -85,B 0,C 180,E1 -31610.382,E2 -31610.382} C_VEL
LIN {X 0,Y 134.358,Z 856.981,A -85,B 0,C 180,E1 -31605.161,E2 -31605.161} C_VEL
LIN {X 0,Y 127.911,Z 859.134,A -85,B 0,C 180,E1 -31598.514,E2 -31598.514} C_VEL
LIN {X 0,Y 123.224,Z 860.098,A -85,B 0,C 180,E1 -31590,E2 -31590} C_VEL
LIN {X 0,Y 127.912,Z 859.133,A -85,B 0,C 180,E1 -31581.484,E2 -31581.484} C_VEL
LIN {X 0,Y 132.001,Z 857.818,A -85,B 0,C 180,E1 -31576.956,E2 -31576.956} C_VEL
LIN {X 0,Y 134.26,Z 857.242,A -85,B 0,C 180,E1 -31575.568,E2 -31575.568} C_VEL
LIN {X 0,Y 144.846,Z 855.049,A -85,B 0,C 180,E1 -31572.252,E2 -31572.252} C_VEL
LIN {X 0,Y 147.308,Z 854.191,A -85,B 0,C 180,E1 -31571.071,E2 -31571.071} C_VEL
LIN {X 0,Y 149.865,Z 853.215,A -85,B 0,C 180,E1 -31569.701,E2 -31569.701} C_VEL
LIN {X 0,Y 154.819,Z 854.177,A -85,B 0,C 180,E1 -31572.417,E2 -31572.417} C_VEL
LIN {X 0,Y 159.892,Z 855.276,A -85,B 0,C 180,E1 -31575.237,E2 -31575.237} C_VEL
LIN {X 0,Y 165.018,Z 856.356,A -85,B 0,C 180,E1 -31578.39,E2 -31578.39} C_VEL
LIN {X 0,Y 167.711,Z 856.977,A -85,B 0,C 180,E1 -31580.351,E2 -31580.351} C_VEL
LIN {X 0,Y 170.866,Z 857.676,A -85,B 0,C 180,E1 -31582.912,E2 -31582.912} C_VEL
LIN {X 0,Y 173.158,Z 858.141,A -85,B 0,C 180,E1 -31585.344,E2 -31585.344} C_VEL
LIN {X 0,Y 175.752,Z 858.448,A -85,B 0,C 180,E1 -31588.571,E2 -31588.571} C_VEL
LIN {X 0,Y 176.167,Z 858.533,A -85,B 0,C 180,E1 -31590,E2 -31590} C_VEL
LIN {X 0,Y 175.752,Z 858.448,A -85,B 0,C 180,E1 -31591.428,E2 -31591.428} C_VEL
LIN {X 0,Y 173.156,Z 858.141,A -85,B 0,C 180,E1 -31594.656,E2 -31594.656} C_VEL
LIN {X 0,Y 170.183,Z 857.548,A -85,B 0,C 180,E1 -31597.647,E2 -31597.647} C_VEL
LIN {X 0,Y 167.7,Z 856.977,A -85,B 0,C 180,E1 -31599.65,E2 -31599.65} C_VEL
LIN {X 0,Y 163.797,Z 856.082,A -85,B 0,C 180,E1 -31602.388,E2 -31602.388} C_VEL
LIN {X 0,Y 158.738,Z 855.039,A -85,B 0,C 180,E1 -31605.405,E2 -31605.405} C_VEL
LIN {X 0,Y 152.578,Z 853.728,A -85,B 0,C 180,E1 -31608.81,E2 -31608.81} C_VEL
LIN {X 0,Y 149.865,Z 853.214,A -85,B 0,C 180,E1 -31610.3,E2 -31610.3} C_VEL
LIN {X 0,Y 148.026,Z 853.869,A -85,B 0,C 180,E1 -31609.411,E2 -31609.411} C_VEL
LIN {X 0,Y 141.35,Z 856.767,A -85,B 0,C 180,E1 -31604.394,E2 -31604.394} C_VEL
LIN {X 0,Y 134.723,Z 859.021,A -85,B 0,C 180,E1 -31597.631,E2 -31597.631} C_VEL
LIN {X 0,Y 130.407,Z 859.886,A -85,B 0,C 180,E1 -31590,E2 -31590} C_VEL
LIN {X 0,Y 134.723,Z 859.021,A -85,B 0,C 180,E1 -31582.367,E2 -31582.367} C_VEL
LIN {X 0,Y 141.349,Z 856.766,A -85,B 0,C 180,E1 -31575.605,E2 -31575.605} C_VEL
LIN {X 0,Y 147.308,Z 854.191,A -85,B 0,C 180,E1 -31571.071,E2 -31571.071} C_VEL
LIN {X 0,Y 147.821,Z 854.43,A -85,B 0,C 180,E1 -31571.614,E2 -31571.614} C_VEL
LIN {X 0,Y 146.902,Z 855.822,A -85,B 0,C 180,E1 -31574.26,E2 -31574.26} C_VEL
LIN {X 0,Y 144.401,Z 857.668,A -85,B 0,C 180,E1 -31578.724,E2 -31578.724} C_VEL
LIN {X 0,Y 142.331,Z 858.658,A -85,B 0,C 180,E1 -31582.113,E2 -31582.113} C_VEL
LIN {X 0,Y 141.497,Z 858.904,A -85,B 0,C 180,E1 -31583.242,E2 -31583.242} C_VEL
LIN {X 0,Y 137.583,Z 859.674,A -85,B 0,C 180,E1 -31590,E2 -31590} C_VEL
LIN {X 0,Y 141.567,Z 858.887,A -85,B 0,C 180,E1 -31596.845,E2 -31596.845} C_VEL
LIN {X 0,Y 148.362,Z 856.552,A -85,B 0,C 180,E1 -31603.701,E2 -31603.701} C_VEL
LIN {X 0,Y 151.005,Z 855.824,A -85,B 0,C 180,E1 -31604.995,E2 -31604.995} C_VEL
LIN {X 0,Y 154.305,Z 856.371,A -85,B 0,C 180,E1 -31603.163,E2 -31603.163} C_VEL
LIN {X 0,Y 159.112,Z 857.237,A -85,B 0,C 180,E1 -31600.176,E2 -31600.176} C_VEL
LIN {X 0,Y 162.947,Z 857.953,A -85,B 0,C 180,E1 -31597.26,E2 -31597.26} C_VEL
LIN {X 0,Y 165.458,Z 858.37,A -85,B 0,C 180,E1 -31594.873,E2 -31594.873} C_VEL
LIN {X 0,Y 168.698,Z 858.686,A -85,B 0,C 180,E1 -31591.063,E2 -31591.063} C_VEL
LIN {X 0,Y 169.037,Z 858.744,A -85,B 0,C 180,E1 -31590,E2 -31590} C_VEL
LIN {X 0,Y 168.698,Z 858.686,A -85,B 0,C 180,E1 -31588.936,E2 -31588.936} C_VEL
LIN {X 0,Y 165.468,Z 858.37,A -85,B 0,C 180,E1 -31585.127,E2 -31585.127} C_VEL
LIN {X 0,Y 162.754,Z 857.914,A -85,B 0,C 180,E1 -31582.557,E2 -31582.557} C_VEL
LIN {X 0,Y 157.616,Z 856.973,A -85,B 0,C 180,E1 -31578.798,E2 -31578.798} C_VEL
LIN {X 0,Y 152.303,Z 856.024,A -85,B 0,C 180,E1 -31575.703,E2 -31575.703} C_VEL
LIN {X 0,Y 151.009,Z 855.821,A -85,B 0,C 180,E1 -31574.999,E2 -31574.999} C_VEL
LIN {X 0,Y 148.362,Z 856.552,A -85,B 0,C 180,E1 -31576.299,E2 -31576.299} C_VEL
LIN {X 0,Y 142.886,Z 858.498,A -85,B 0,C 180,E1 -31581.515,E2 -31581.515} C_VEL
LIN {X 0,Y 141.497,Z 858.904,A -85,B 0,C 180,E1 -31583.242,E2 -31583.242} C_VEL
LIN {X 0,Y 140.972,Z 859.204,A -85,B 0,C 180,E1 -31584.819,E2 -31584.819} C_VEL
LIN {X 0,Y 141.475,Z 859.361,A -85,B 0,C 180,E1 -31586.418,E2 -31586.418} C_VEL
LIN {X 0,Y 145.201,Z 859.391,A -85,B 0,C 180,E1 -31591.077,E2 -31591.077} C_VEL
LIN {X 0,Y 145.503,Z 859.346,A -85,B 0,C 180,E1 -31591.601,E2 -31591.601} C_VEL
LIN {X 0,Y 150.091,Z 858.286,A -85,B 0,C 180,E1 -31598.075,E2 -31598.075} C_VEL
LIN {X 0,Y 152.643,Z 857.897,A -85,B 0,C 180,E1 -31599.11,E2 -31599.11} C_VEL
LIN {X 0,Y 155.708,Z 858.354,A -85,B 0,C 180,E1 -31596.796,E2 -31596.796} C_VEL
LIN {X 0,Y 157.6,Z 858.605,A -85,B 0,C 180,E1 -31595.117,E2 -31595.117} C_VEL
LIN {X 0,Y 160.056,Z 858.85,A -85,B 0,C 180,E1 -31592.517,E2 -31592.517} C_VEL
LIN {X 0,Y 161.652,Z 858.924,A -85,B 0,C 180,E1 -31590.667,E2 -31590.667} C_VEL
LIN {X 0,Y 161.902,Z 858.955,A -85,B 0,C 180,E1 -31590,E2 -31590} C_VEL
LIN {X 0,Y 161.652,Z 858.924,A -85,B 0,C 180,E1 -31589.333,E2 -31589.333} C_VEL
LIN {X 0,Y 160.06,Z 858.85,A -85,B 0,C 180,E1 -31587.483,E2 -31587.483} C_VEL
LIN {X 0,Y 157.621,Z 858.605,A -85,B 0,C 180,E1 -31584.884,E2 -31584.884} C_VEL
LIN {X 0,Y 154.299,Z 858.162,A -85,B 0,C 180,E1 -31582.147,E2 -31582.147} C_VEL
LIN {X 0,Y 152.637,Z 857.893,A -85,B 0,C 180,E1 -31580.88,E2 -31580.88} C_VEL
LIN {X 0,Y 150.051,Z 858.287,A -85,B 0,C 180,E1 -31581.923,E2 -31581.923} C_VEL
LIN {X 0,Y 146.119,Z 859.262,A -85,B 0,C 180,E1 -31587.243,E2 -31587.243} C_VEL
LIN {X 0,Y 144.756,Z 859.462,A -85,B 0,C 180,E1 -31590,E2 -31590} C_VEL
LIN {X 0,Y 145.503,Z 859.346,A -85,B 0,C 180,E1 -31591.601,E2 -31591.601} C_VEL
LIN {X 0,Y 146.526,Z 859.323,A -85,B 0,C 180,E1 -31591.602,E2 -31591.602} C_VEL
LIN {X 0,Y 148.152,Z 859.319,A -85,B 0,C 180,E1 -31590.974,E2 -31590.974} C_VEL
LIN {X 0,Y 153.069,Z 859.122,A -85,B 0,C 180,E1 -31588.34,E2 -31588.34} C_VEL
LIN {X 0,Y 153.337,Z 859.108,A -85,B 0,C 180,E1 -31588.319,E2 -31588.319} C_VEL
LIN {X 0,Y 151.928,Z 859.25,A -85,B 0,C 180,E1 -31590,E2 -31590} C_VEL
LIN {X 0,Y 153.337,Z 859.108,A -85,B 0,C 180,E1 -31591.677,E2 -31591.677} C_VEL
LIN {X 0,Y 154.742,Z 859.167,A -85,B 0,C 180,E1 -31590,E2 -31590} C_VEL
LIN {X 0,Y 153.337,Z 859.108,A -85,B 0,C 180,E1 -31588.319,E2 -31588.319} C_VEL
LIN {X 0,Y 153.337,Z 859.108,A -85,B 0,C 180,E1 -31588.319,E2 -31588.319}

QRS_NEXT_CUT()

QRS_NEXT()
QRS_HOME()

END
